(* CODESYS project testSpiIO.project

Project tree, tasks and I/O mapping:
  Device : Jinan Cherry-ARM Cortex-VxWorks, Jinan Cheery Electric Co., Ltd., version 3.5.11.20
    application Application
      libraries: Standard, * (System)
      task MainTask (cyclic, interval 500 ms, priority 1) calls PLC_PRG
      program PLC_PRG [ST]
    SoftMotion General Axis Pool
    IoDrvSOC : IoDrvSOC, Hitech, version 1.0.0.0
        unmapped channels: in1, in2, in3, in4, in5, in6, in7, in8, out1, out2, out3, out4, out5, out6, out7, out8
    IoDrvSpiIO : IoDrvSpiIO, Hitech, version 1.0.0.0
        input  Application.PLC_PRG.sDI[1] : BOOL  // spi1in1
        input  Application.PLC_PRG.sDI[2] : BOOL  // spi1in2
        input  Application.PLC_PRG.sDI[3] : BOOL  // spi1in3
        input  Application.PLC_PRG.sDI[4] : BOOL  // spi1in4
        input  Application.PLC_PRG.sDI[5] : BOOL  // spi1in5
        input  Application.PLC_PRG.sDI[6] : BOOL  // spi1in6
        input  Application.PLC_PRG.sDI[7] : BOOL  // spi1in7
        input  Application.PLC_PRG.sDI[8] : BOOL  // spi1in8
        input  Application.PLC_PRG.sDI[9] : BOOL  // spi1in9
        input  Application.PLC_PRG.sDI[10] : BOOL  // spi1in10
        input  Application.PLC_PRG.sDI[11] : BOOL  // spi1in11
        input  Application.PLC_PRG.sDI[12] : BOOL  // spi1in12
        input  Application.PLC_PRG.sDI[13] : BOOL  // spi1in13
        input  Application.PLC_PRG.sDI[14] : BOOL  // spi1in14
        input  Application.PLC_PRG.sDI[15] : BOOL  // spi1in15
        input  Application.PLC_PRG.sDI[16] : BOOL  // spi1in16
        input  Application.PLC_PRG.sDI[17] : BOOL  // spi2in1
        input  Application.PLC_PRG.sDI[18] : BOOL  // spi2in2
        input  Application.PLC_PRG.sDI[19] : BOOL  // spi2in3
        input  Application.PLC_PRG.sDI[20] : BOOL  // spi2in4
        input  Application.PLC_PRG.sDI[21] : BOOL  // spi2in5
        input  Application.PLC_PRG.sDI[22] : BOOL  // spi2in6
        input  Application.PLC_PRG.sDI[23] : BOOL  // spi2in7
        input  Application.PLC_PRG.sDI[24] : BOOL  // spi2in8
        input  Application.PLC_PRG.sDI[25] : BOOL  // spi2in9
        input  Application.PLC_PRG.sDI[26] : BOOL  // spi2in10
        input  Application.PLC_PRG.sDI[27] : BOOL  // spi2in11
        input  Application.PLC_PRG.sDI[28] : BOOL  // spi2in12
        output Application.PLC_PRG.sDO[1] : BOOL  // spi1out1
        output Application.PLC_PRG.sDO[2] : BOOL  // spi1out2
        output Application.PLC_PRG.sDO[3] : BOOL  // spi1out3
        output Application.PLC_PRG.sDO[4] : BOOL  // spi1out4
        output Application.PLC_PRG.sDO[5] : BOOL  // spi1out5
        output Application.PLC_PRG.sDO[6] : BOOL  // spi1out6
        output Application.PLC_PRG.sDO[7] : BOOL  // spi1out7
        output Application.PLC_PRG.sDO[8] : BOOL  // spi1out8
        output Application.PLC_PRG.sDO[9] : BOOL  // spi1out9
        output Application.PLC_PRG.sDO[10] : BOOL  // spi1out10
        output Application.PLC_PRG.sDO[11] : BOOL  // spi1out11
        output Application.PLC_PRG.sDO[12] : BOOL  // spi1out12
        output Application.PLC_PRG.sDO[13] : BOOL  // spi1out13
        output Application.PLC_PRG.sDO[14] : BOOL  // spi1out14
        output Application.PLC_PRG.sDO[15] : BOOL  // spi1out15
        output Application.PLC_PRG.sDO[16] : BOOL  // spi1out16
        output Application.PLC_PRG.sDO[17] : BOOL  // spi2out1
        output Application.PLC_PRG.sDO[18] : BOOL  // spi2out2
        output Application.PLC_PRG.sDO[19] : BOOL  // spi2out3
        output Application.PLC_PRG.sDO[20] : BOOL  // spi2out4
        output Application.PLC_PRG.sDO[21] : BOOL  // spi2out5
        output Application.PLC_PRG.sDO[22] : BOOL  // spi2out6
        output Application.PLC_PRG.sDO[23] : BOOL  // spi2out7
        output Application.PLC_PRG.sDO[24] : BOOL  // spi2out8
        output Application.PLC_PRG.sDO[25] : BOOL  // spi2out9
        output Application.PLC_PRG.sDO[26] : BOOL  // spi2out10
        output Application.PLC_PRG.sDO[27] : BOOL  // spi2out11
        output Application.PLC_PRG.sDO[28] : BOOL  // spi2out12
        output Application.PLC_PRG.sDO[29] : BOOL  // spi2out13
        output Application.PLC_PRG.sDO[30] : BOOL  // spi2out14
        output Application.PLC_PRG.sDO[31] : BOOL  // spi2out15
        output Application.PLC_PRG.sDO[32] : BOOL  // spi2out16
*)

// Device/Application/PLC_PRG
PROGRAM PLC_PRG
VAR	
	sDO : ARRAY[1..32] OF BOOL;
	//hDO : ARRAY[1..6] OF BOOL;
	sDI : ARRAY[1..28] OF BOOL;
	i : INT;
	init : BOOL := FALSE;
	init2 : BOOL := FALSE;
END_VAR

IF init = FALSE THEN	
	FOR i := 1 TO 32 BY +1 DO
		sDO[i] := false; //SET HIGH
	END_FOR	
	init := TRUE;
END_IF

(*
FOR i := 24 TO 17 BY -1 DO
	sDO[i] := TRUE;  //SET HIGH
END_FOR
*)

END_PROGRAM
